// TwinCAT 3 PLC project RectangleSlicingMachine
// ProgramVersion: 3.1.4024.0
// libraries:
//   Tc2_MC2, * (Beckhoff Automation GmbH)
//   Tc2_NC, * (Beckhoff Automation GmbH)
//   Tc2_Standard, * (Beckhoff Automation GmbH)
//   Tc2_System, * (Beckhoff Automation GmbH)
//   Tc3_Module, * (Beckhoff Automation GmbH)
//   VisuDialogs, * (System)
// project tree:
//   / GlobalTextList.TcGTLO, PlcTask.TcTTO (not stored), Visualization Manager.TcVMO (not stored)
//   POUs/ FB_Slicer.TcPOU, MAIN.TcPOU, PRG_Test.TcPOU
//   VISUs/ Visualization.TcVIS
// real-time tasks:
//   TASK PlcTask: cycle T#10ms, priority 20, ADS port 350
// motion (NC):
//   TASK NC-Task 1 SAF: cycle T#2ms, priority 4, ADS port 501
//   TASK NC-Task 1 SVB: cycle T#10ms, priority 8, ADS port 511
//   AXIS AxisM1 (id 1)
//     General: UnitName=Degree
//     Velo: Maximum=18000
//     OtherSettings: AllowMotionCmdToSlave=true
//     encoder EncType=1
//     drive DrvType=5
//       Analog: TorqueSetpointScale=10, ScaleFactorActTorque=0.1
//       TimeComp: TaskDelayCycles=1
//     controller CtrType=1
//       CtrPara: PriorControlFactor=1
//         Observer: BandWidth=20
//   AXIS AxisM1s (id 2)
//     General: UnitName=Degree
//     Velo: Maximum=18000
//     OtherSettings: AllowMotionCmdToSlave=true
//     encoder EncType=1
//     drive DrvType=5
//       Analog: TorqueSetpointScale=10, ScaleFactorActTorque=0.1
//       TimeComp: TaskDelayCycles=1
//     controller CtrType=1
//       CtrPara: PriorControlFactor=1
//         Observer: BandWidth=20
//   AXIS AxisM2 (id 3)
//     General: UnitName=Degree
//     Velo: Maximum=18000
//     OtherSettings: AllowMotionCmdToSlave=true
//     encoder EncType=1
//     drive DrvType=5
//       Analog: TorqueSetpointScale=10, ScaleFactorActTorque=0.1
//       TimeComp: TaskDelayCycles=1
//     controller CtrType=1
//       CtrPara: PriorControlFactor=1
//         Observer: BandWidth=20
//   AXIS Axis 4 (id 4)
//     General: UnitName=°
//     Dynamic: Acceleration=12000, Deceleration=12000, Jerk=114759
//     Velo: Maximum=18000
//     PositionAreaControl: Enable=false
//     TargetPosControl: Enable=false
//     OtherSettings: AllowMotionCmdToSlave=true
//     encoder EncType=19
//       EncPara: ScaleFactorNumerator=360, ScaleFactorDenominator=65536, MaxCount=#xffffffff
//     drive DrvType=16
//       DrvPara: MaxCount=#xffffffff, DriveControlDWord=#x00020100
//         Analog: VeloReferenz=18000, TorqueSetpointScale=10, ScaleFactorActTorque=0.1
//         TimeComp: TaskDelayCycles=1
//     controller CtrType=1
//       CtrPara: PriorControlFactor=1
//         PosDiffControl: Enable=false
//         Observer: BandWidth=20
// I/O:
//   DEVICE Device 1 (EtherCAT) (disabled), AmsNetId 10.0.20.72.2.1
//     Drive 1 (i950 (BS-STO)) [i950 (BS-STO) FW V01.09]
//       modules: Module 1 (Universal (CSP + Speed and Torque Limits))
//     Drive 2 (i950 (BS-STO)) [i950 (BS-STO) FW V01.09]
//       modules: Module 1 (Universal (CSP + Speed and Torque Limits))
// variable links:
//   RectangleSlicingMachine/RectangleSlicingMachine Instance <-> Device 1 (EtherCAT)/Drive 1 (i950 (BS-STO))
//     PlcTask Outputs/MAIN.fbSlicer.nDrive1NegativeTorqueLimit <-> Module 1 (Universal (CSP + Speed and Torque Limits))/Torque Limits/MAIN.fbSlicer.nDrive1NegativeTorqueLimit
//     PlcTask Outputs/MAIN.fbSlicer.nDrive1PositiveTorqueLimit <-> Module 1 (Universal (CSP + Speed and Torque Limits))/Torque Limits/MAIN.fbSlicer.nDrive1PositiveTorqueLimit
//   RectangleSlicingMachine/RectangleSlicingMachine Instance <-> Device 1 (EtherCAT)/Drive 2 (i950 (BS-STO))
//     PlcTask Outputs/MAIN.fbSlicer.nDrive2NegativeTorqueLimit <-> Module 1 (Universal (CSP + Speed and Torque Limits))/Torque Limits/MAIN.fbSlicer.nDrive2NegativeTorqueLimit
//     PlcTask Outputs/MAIN.fbSlicer.nDrive2PositiveTorqueLimit <-> Module 1 (Universal (CSP + Speed and Torque Limits))/Torque Limits/MAIN.fbSlicer.nDrive2PositiveTorqueLimit
//   RectangleSlicingMachine/RectangleSlicingMachine Instance <-> NC-Task 1 SAF/Axes/AxisM1
//     PlcTask Inputs/MAIN.fbSlicer.AxisM1.NcToPlc <-> Outputs/ToPlc
//     PlcTask Outputs/MAIN.fbSlicer.AxisM1.PlcToNc <-> Inputs/FromPlc
//   RectangleSlicingMachine/RectangleSlicingMachine Instance <-> NC-Task 1 SAF/Axes/AxisM1s
//     PlcTask Inputs/MAIN.fbSlicer.AxisM1s.NcToPlc <-> Outputs/ToPlc
//     PlcTask Outputs/MAIN.fbSlicer.AxisM1s.PlcToNc <-> Inputs/FromPlc
//   RectangleSlicingMachine/RectangleSlicingMachine Instance <-> NC-Task 1 SAF/Axes/AxisM2
//     PlcTask Inputs/MAIN.fbSlicer.AxisM2.NcToPlc <-> Outputs/ToPlc
//     PlcTask Outputs/MAIN.fbSlicer.AxisM2.PlcToNc <-> Inputs/FromPlc

// ---- POUs/FB_Slicer.TcPOU
FUNCTION_BLOCK FB_Slicer
VAR_INPUT
	// Buttons to control various actions
	bStartButton : BOOL;
	bStopButton : BOOL;
	bContinueButton : BOOL;
	bHomeButton: BOOL;	// Returns axes to 0
	bEnginesOnButton : BOOL;
	bEnginesOffButton : BOOL;
	
	// Coordinates for the slicing start position
	aStartingPosition : ARRAY[0..1] OF LREAL;
	// Dimensions of the rectangle to be sliced
	aSlicingDimensions : ARRAY[0..1] OF LREAL;
	
	// Velocity override for motor movements
	fVelocityOverride : LREAL;
END_VAR
VAR_OUTPUT
	// Current positions of motors M1, M1s and M2
	fM1Position : LREAL;
	fM1sPosition : LREAL;
	fM2Position : LREAL;
	
	//Lights
	bEnginesLight : BOOL;	// On when the engines are on
	bHomedLight : BOOL;		// On when the axes are homed
	bSlicingLight : BOOL;	// On when slicing is happening
	bStopLight : BOOL;		// On when the process is stopped
	bErrorLight : BOOL;		// On when there's an error
	
	nErrorID : UDINT;
END_VAR
VAR
	// Trigger functions to stop bouncing when any of the buttons are pressed
	fbStartButtonTrigger : R_TRIG;
	fbStopButtonTrigger : R_TRIG;
	fbContinueButtonTrigger : R_TRIG;
	fbHomeButtonTrigger : R_TRIG;
	fbEnginesOnButtonTrigger : R_TRIG;
	fbEnginesOffButtonTrigger : R_TRIG;
	
	// References to the axes
	AxisM1 : AXIS_REF;	// Master
	AxisM1s : AXIS_REF;	// Slave
	AxisM2 : AXIS_REF;
	
	// Adequate function blocks needed for the axes
	M1McPower : MC_Power;
	M1McMoveRelative : MC_MoveRelative;
	M1McHome : MC_Home;
	M1McReset : MC_Reset;
	M1McStop : MC_Stop;
	
	M1sMcPower : MC_Power;
	M1sMcMoveRelative : MC_MoveRelative;
	M1sMcHome : MC_Home;
	M1sMcSetPosition : MC_SetPosition;
	M1sMcReset : MC_Reset;
	M1sMcStop : MC_Stop;
	
	M2McPower : MC_Power;
	M2McMoveRelative : MC_MoveRelative;
	M2McHome : MC_Home;
	M2McReset : MC_Reset;
	M2McStop : MC_Stop;
	
	// FBs needed to synchronise and desynchronize M1s to M1
	McGearIn : MC_GearIn;
	McGearOut : MC_GearOut;
	
	// Variable to tell us if the axes are homed or not
	bHomed : BOOL;
	
	// Variable to tell us if the engines are on or off (TRUE - ON, FALSE - OFF)
	bPowerStatus : BOOL;
	
	// Variable to tell us if M1 and M1s are coupled or not
	bCoupled  : BOOL;
	
	// Variable to tell us if the return button is pressed
	bReturned : BOOL;
	
	(* Variable to tell us if the user has given all coordinates needed (starting position and
	   rectangle dimensions) in order for the machine to be able to start *)
	bCoordinates : BOOL;
	
	// Variable to tell us if the dimensions we've given make the machine go out of bounds
	bLimit : BOOL;
	
	// Slicing dimensions 
	fM1SlicingDistance : LREAL;
	fM2SlicingDistance : LREAL;
	// Starting point dimensions
	fM1StartingDistance : LREAL;
	fM2StartingDistance : LREAL;
	
	// Variables used to keep track of the state in which we stopped and update the dimensions
	nStoppedState : DINT;
	fTempM1SlicingDistance : LREAL;
	fTempM2SlicingDistance : LREAL;
	fTempM1StartingDistance : LREAL;
	fTempM2StartingDistance : LREAL;

	
	// Variable needed for initializing the CASE structure states
	nCurrentState : DINT;
	
	// Needed torques for the I/O
	nDrive1PositiveTorqueLimit AT %Q* : INT := 1000;
    nDrive1NegativeTorqueLimit AT %Q* : INT := 1000;
    nDrive2PositiveTorqueLimit AT %Q* : INT := 1000;
    nDrive2NegativeTorqueLimit AT %Q* : INT := 1000;
	
END_VAR

VAR CONSTANT
	// Define limits
	MINIMUM_STARTING_POSITION : UINT := 10;
	MAXIMUM_SLICING_DIMENSION : UINT := 80;
END_VAR

(* This FB deals with controlling a machine that's got 3 motors with incremental encoders. Two of them (M1 & M1s) 
   function synchronous moving a slicer on the y axis whereas the third one (M2) moves the slicer on the x axis. 
   M1 & M1s have a master - slave configuration. The idea is that the machine will be used to cut rectangles with 
   dimensions given by the user, so what we want to do is to home the axes, take the slicer to a predefined 
   position where we want the slicing to start and cut out a rectangle by moving M1 & M1s synchronously positive 
   the y axis, then M2 in a positive direction on the x axis, then M1 & M1s negative y and then M2 negative x. 
   The machine operates within a 100x100cm workspace, which necessitates setting boundaries to avoid exceeding the 
   machine's limits. To ensure a safe margin, I've established a 10 cm buffer on all sides. So, the minimum starting
   position for any operation is (10,10) cm. Based on this configuration, the largest rectangle the machine can 
   safely cut is 80x80cm without crossing the predefined boundaries.*)
   
   
CASE nCurrentState OF
	0:	// Power OFF
	bEnginesLight := FALSE;
	bPowerStatus := FALSE;

	M1McPower.Enable := FALSE;
	M1McPower.Enable_Positive := FALSE;
	M1McPower.Enable_Negative := FALSE;
	M1McPower.Override := fVelocityOverride;
	
	M1sMcPower.Enable := FALSE;
	M1sMcPower.Enable_Positive := FALSE;
	M1sMcPower.Enable_Negative := FALSE;
	M1sMcPower.Override := fVelocityOverride;
	
	M2McPower.Enable := FALSE;
	M2McPower.Enable_Positive := FALSE;
	M2McPower.Enable_Negative := FALSE;
	M2McPower.Override := fVelocityOverride;
	  
	IF bEnginesOnButton THEN
		nCurrentState := 10;
	END_IF
	
	10:	// Power ON
	bEnginesLight := TRUE;
	bPowerStatus := TRUE;
	
	M1McPower.Enable := TRUE;
	M1McPower.Enable_Positive := TRUE;
	M1McPower.Enable_Negative := TRUE;
	M1McPower.Override := fVelocityOverride;
	
	M1sMcPower.Enable := TRUE;
	M1sMcPower.Enable_Positive := TRUE;
	M1sMcPower.Enable_Negative := TRUE;
	M1sMcPower.Override := fVelocityOverride;
	
	M2McPower.Enable := TRUE;
	M2McPower.Enable_Positive := TRUE;
	M2McPower.Enable_Negative := TRUE;
	M2McPower.Override := fVelocityOverride;
		  
	IF M1McPower.Active AND M1sMcPower.Active AND M2McPower.Active THEN
		nCurrentState := 25;
	END_IF		  

	25:	// Reseting
	bSlicingLight := FALSE;
	bStopLight := FALSE;
	
	// Reset the axes
	M1McReset.Execute := TRUE;
	IF NOT bCoupled THEN
		M1sMcReset.Execute := TRUE;
		IF M1sMcReset.Done THEN
			M1sMcReset.Execute := FALSE;
		END_IF
	END_IF
	M2McReset.Execute := TRUE;
	
	// If the reseting is done, go check if the axes are ready for operation
	IF M1McReset.Done AND M2McReset.Done THEN
		M1McReset.Execute := FALSE;	
		M2McReset.Execute := FALSE;
		
		//IF nStoppedState = 200 OR nStoppedState = 300 OR nStoppedState = 400 OR nStoppedState = 500 OR nStoppedState = 600 OR nStoppedState = 650 THEN
		//	nCurrentState := nStoppedState;
		//ELSE
		//	nCurrentState := 50;
		//END_IF
		
		nCurrentState := 50;
		
	END_IF
	
	// Check for errors during the reseting
	IF M1McReset.Error THEN
		nErrorID := M1McReset.ErrorID;
		nCurrentState := 999;
	END_IF
	IF M1sMcReset.Error THEN
		nErrorID := M1sMcReset.ErrorID;
		nCurrentState := 999;
	END_IF
	IF M2McReset.Error THEN
		nErrorID := M2McReset.ErrorID;
		nCurrentState := 999;
	END_IF

	50: // Checking if the axes are ready for operation
	IF M1McPower.Status AND M1sMcPower.Status AND M2McPower.Status AND bPowerStatus THEN
		nCurrentState := 75;
	END_IF	
	
	// If there is some error go to the error state
	IF M1McPower.Error THEN
		nErrorID := M1McPower.ErrorID;
		nCurrentState := 999;
	END_IF
	IF M1sMcPower.Error THEN
		nErrorID := M1sMcPower.ErrorID;
		nCurrentState := 999;
	END_IF
	IF M2McPower.Error THEN
		nErrorID := M2McPower.ErrorID;
		nCurrentState := 999;
	END_IF
	
	75:		// Setting the slave axis to 0
		M1sMcSetPosition.Execute := TRUE;
		M1sMcSetPosition.Position := 0;
					 
		IF M1sMcSetPosition.Done THEN
			M1sMcSetPosition.Execute := FALSE;
			nCurrentState := 100;
		END_IF

	100:	// Gearing
	// Synchronize M1s to M1. The ratio is 1 because they have to move synchronously
	McGearIn.Execute := TRUE;
	McGearIn.RatioNumerator := 1;
	McGearIn.RatioDenominator := 1;
		
	// If they're coupled go to homing
	IF McGearIn.InGear THEN
		bCoupled := TRUE;
		
		IF nStoppedState = 200 OR nStoppedState = 300 OR nStoppedState = 400 OR nStoppedState = 500 OR nStoppedState = 600 OR nStoppedState = 650 THEN
			nCurrentState := nStoppedState;
		ELSE
			nCurrentState := 150;
		END_IF
		
		//nCurrentState := 150;
	END_IF
	
	150:	// Homing
	// Home the axes with incremental encoders to 0
	M1McHome.Execute := TRUE;
	M1McHome.Position := 0;
	M1McHome.HomingMode := MC_Direct;
	
	M2McHome.Execute := TRUE;
	M2McHome.Position := 0;
	M2McHome.HomingMode := MC_Direct;
				 
	// If the homing is done, stop executing it
	IF M1McHome.Done AND M2McHome.Done THEN
		M1McHome.Execute := FALSE;
		M2McHome.Execute := FALSE;
	END_IF
	
	// If there is some error go to the error state
	IF M1McHome.Error THEN
		nErrorID := M1McHome.ErrorID;
		nCurrentState := 999;
	END_IF
	IF M2McHome.Error THEN
		nErrorID := M2McHome.ErrorID;
		nCurrentState := 999;
	END_IF
				
	// If the start button is pressed and the given coordinates are valid go to the slicing starting position 
	IF bStartButton AND bCoordinates THEN
		nCurrentState := 200;
	END_IF
	
	200:	// Slicing starting position
	IF nStoppedState = 200 THEN
		nStoppedState := 0;
		fM1StartingDistance := fTempM1StartingDistance;
		fM2StartingDistance := fTempM2StartingDistance;
	ELSE
		fTempM1StartingDistance := aStartingPosition[0];
		fTempM2StartingDistance := aStartingPosition[1];
	END_IF
	
	// Move all motors to the starting position
	M1McMoveRelative.Execute := TRUE;
	M1McMoveRelative.Distance := fTempM1StartingDistance;
	M1McMoveRelative.Velocity := 10;
	M1McMoveRelative.Acceleration := 10;
	M1McMoveRelative.Deceleration := 10;
	M1McMoveRelative.Jerk := 10000;
					 
	M2McMoveRelative.Execute := TRUE;
	M2McMoveRelative.Distance := fTempM2StartingDistance;
	M2McMoveRelative.Velocity := 10;
	M2McMoveRelative.Acceleration := 10;
	M2McMoveRelative.Deceleration := 10;
	M2McMoveRelative.Jerk := 10000;
					 
	// If all motors reach the starting position go to the first slicing state
	IF M1McMoveRelative.Done AND M2McMoveRelative.Done THEN
		M1McMoveRelative.Execute := FALSE;
		M2McMoveRelative.Execute := FALSE;
		
		nCurrentState := 300;
	END_IF
	
	// If error -> go to error state
	IF M1McMoveRelative.Error OR M2McMoveRelative.Error THEN
		IF M1McMoveRelative.Error THEN
			nErrorID := M1McMoveRelative.ErrorID;
		ELSIF M2McMoveRelative.Error THEN
			nErrorID := M2McMoveRelative.ErrorID;
		END_IF
		nCurrentState := 999;
	END_IF
					 
	300:	// Moving M1 & M1s positive y
	bSlicingLight := TRUE;
	
	IF nStoppedState = 300 THEN
		nStoppedState := 0;
		fM1SlicingDistance := fTempM1SlicingDistance;
	ELSE
		fM1SlicingDistance := aSlicingDimensions[0];
	END_IF
	
	M1McMoveRelative.Execute := TRUE;
	M1McMoveRelative.Distance := fM1SlicingDistance;
	M1McMoveRelative.Velocity := 5;
	M1McMoveRelative.Acceleration := 5;
	M1McMoveRelative.Deceleration := 5;
	M1McMoveRelative.Jerk := 10000;
				
	// If the moving is done, move on to the next	
	IF M1McMoveRelative.Done THEN
		M1McMoveRelative.Execute := FALSE;
		nCurrentState := 400;
	END_IF
	
	// If error -> go to error state
	IF M1McMoveRelative.Error THEN
		nErrorID := M1McMoveRelative.ErrorID;
		nCurrentState := 999;
	END_IF
	
	400:	// Moving M2 positive x
	bSlicingLight := TRUE;
	
	IF nStoppedState = 400 THEN
		nStoppedState := 0;
		fM2SlicingDistance := fTempM2SlicingDistance;
	ELSE
		fM2SlicingDistance := aSlicingDimensions[1];
	END_IF
	
	M2McMoveRelative.Execute := TRUE;
	M2McMoveRelative.Distance := fM2SlicingDistance;
	M2McMoveRelative.Velocity := 10;
	M2McMoveRelative.Acceleration := 10;
	M2McMoveRelative.Deceleration := 10;
	M2McMoveRelative.Jerk := 10000;
				
	// If the moving is done, move on to the next	
	IF M2McMoveRelative.Done THEN
		M2McMoveRelative.Execute := FALSE;
		nCurrentState := 500;
	END_IF
	
	// If error -> go to error state
	IF M2McMoveRelative.Error THEN
		nErrorID := M2McMoveRelative.ErrorID;
		nCurrentState := 999;
	END_IF
	
	500:	// Moving M1 & M1s negative y
	bSlicingLight := TRUE;
	
	IF nStoppedState = 500 THEN
		nStoppedState := 0;
		fM1SlicingDistance := fTempM1SlicingDistance;
	ELSE
		fM1SlicingDistance := aSlicingDimensions[0];
	END_IF
	
	M1McMoveRelative.Execute := TRUE;
	M1McMoveRelative.Distance := -fM1SlicingDistance;
	M1McMoveRelative.Velocity := 5;
	M1McMoveRelative.Acceleration := 5;
	M1McMoveRelative.Deceleration := 5;
	M1McMoveRelative.Jerk := 10000;
				
	// If the moving is done, move on to the next	
	IF M1McMoveRelative.Done THEN
		M1McMoveRelative.Execute := FALSE;
		nCurrentState := 600;
	END_IF
	
	// If error -> go to error state
	IF M1McMoveRelative.Error THEN
		nErrorID := M1McMoveRelative.ErrorID;
		nCurrentState := 999;
	END_IF
	
	600:	// Moving M2 negative x
	bSlicingLight := TRUE;
	
	IF nStoppedState = 600 THEN
		nStoppedState := 0;
		fM2SlicingDistance := fTempM2SlicingDistance;
	ELSE
		fM2SlicingDistance := aSlicingDimensions[1];
	END_IF
	
	M2McMoveRelative.Execute := TRUE;
	M2McMoveRelative.Distance := -fM2SlicingDistance;
	M2McMoveRelative.Velocity := 10;
	M2McMoveRelative.Acceleration := 10;
	M2McMoveRelative.Deceleration := 10;
	M2McMoveRelative.Jerk := 10000;
	
	// If the moving is done it means the rectangle is cut -> go to (0,0) position
	IF M2McMoveRelative.Done THEN
		M2McMoveRelative.Execute := FALSE;
		nCurrentState := 650;
	END_IF
	
	// If error -> go to error state
	IF M2McMoveRelative.Error THEN
		nErrorID := M2McMoveRelative.ErrorID;
		nCurrentState := 999;
	END_IF
	
	650:	// Return the axes to position (0,0)
	M1McMoveRelative.Execute := TRUE;
    M1McMoveRelative.Distance := -fM1Position;

    M2McMoveRelative.Execute := TRUE;
    M2McMoveRelative.Distance := -fM2Position;
	
	// If the axes are returned -> go to decouple the axes
	IF M1McMoveRelative.Done AND M2McMoveRelative.Done THEN
		M1McMoveRelative.Execute := FALSE;
		M2McMoveRelative.Execute := FALSE;
		nCurrentState := 700;
	END_IF
	
	// If error -> go to error state
	IF M1McMoveRelative.Error OR M2McMoveRelative.Error THEN
		IF M1McMoveRelative.Error THEN
			nErrorID := M1McMoveRelative.ErrorID;
		ELSIF M2McMoveRelative.Error THEN
			nErrorID := M2McMoveRelative.ErrorID;
		END_IF
		nCurrentState := 999;
	END_IF
	
	700:	// Decouple the axes
	McGearIn.Execute := FALSE;
			 
	McGearOut.Execute := TRUE;
			  
	// If the decoupling is done, move to the initial state
	IF McGearOut.Done THEN
		bCoupled := FALSE;
		McGearOut.Execute := FALSE;
				  
		IF NOT bEnginesLight THEN
			nCurrentState := 0;	  
		ELSE
			nCurrentState := 25;
		END_IF
	END_IF
	
	800:	// Stop	
	bSlicingLight := FALSE;
	bStopLight := TRUE;
	
	M1McStop.Execute := TRUE;
	M1McStop.Deceleration := 10;
	M1McStop.Jerk := 10000;
	
	M2McStop.Execute := TRUE;
	M2McStop.Deceleration := 10;
	M2McStop.Jerk := 10000;
			 
	IF M1McStop.Done THEN
		M1McStop.Execute := FALSE;
	END_IF
	
	IF M2McStop.Done THEN
		M2McStop.Execute := FALSE;
	END_IF
	
	// If we press on the continue button we want to continue where we left off
	IF bContinueButton THEN
		(* Since we are using incremental encoders and hence relative movements, we need 
		   to do some math to determine the distance the slicer should go to. We'll give these 
		   values as  dimensions of the rectangle or coordinates of the starting position. *)
		IF nStoppedState = 200 THEN
			fTempM1StartingDistance := aStartingPosition[0] - fM1Position;
			fTempM2StartingDistance := aStartingPosition[1] - fM2Position;
		ELSIF nStoppedState = 300 THEN
			fTempM1SlicingDistance := aStartingPosition[0] + aSlicingDimensions[0] - fM1Position;
		ELSIF nStoppedState = 400 THEN
			fTempM2SlicingDistance := aStartingPosition[1] + aSlicingDimensions[1] - fM2Position;
		ELSIF nStoppedState = 500 THEN
			fTempM1SlicingDistance := fM1Position - aStartingPosition[0];
		ELSIF nStoppedState = 600 THEN
			fTempM2SlicingDistance := fM2Position - aStartingPosition[1];
		END_IF
		
		nCurrentState := 700;	// Reseting must be done after stopping the axes
	END_IF
	
	IF bHomeButton THEN
		nStoppedState := 650;
		nCurrentState := 700;
	END_IF
	
	999:	// Error
	bErrorLight := TRUE;
	
	M1McStop.Execute := TRUE;
	M1McStop.Deceleration := 10;
	M1McStop.Jerk := 10000;
	
	M2McStop.Execute := TRUE;
	M2McStop.Deceleration := 10;
	M2McStop.Jerk := 10000;
			 
	IF M1McStop.Done THEN
		M1McStop.Execute := FALSE;
	END_IF
	
	IF M2McStop.Done THEN
		M2McStop.Execute := FALSE;
	END_IF
	
	ADSLOGDINT(msgCtrlMask := ADSLOG_MSGTYPE_ERROR,
			   msgFmtStr := TO_STRING(nErrorID),
			   dintArg := 0);
			   
	// If the start button is pressed go to the reset state 
	IF bStartButton THEN
		bErrorLight := FALSE;
		nCurrentState := 25;
	END_IF
END_CASE

// Trigger logic
fbStartButtonTrigger(CLK := bStartButton);
bStartButton := fbStartButtonTrigger.Q;
fbStopButtonTrigger(CLK := bStopButton);
bStopButton := fbStopButtonTrigger.Q;
fbContinueButtonTrigger(CLK := bContinueButton);
bContinueButton := fbContinueButtonTrigger.Q;
fbHomeButtonTrigger(CLK := bHomeButton);
bHomeButton := fbHomeButtonTrigger.Q;
fbEnginesOnButtonTrigger(CLK := bEnginesOnButton);
bEnginesOnButton := fbEnginesOnButtonTrigger.Q;
fbEnginesOffButtonTrigger(CLK := bEnginesOffButton);
bEnginesOffButton := fbEnginesOffButtonTrigger.Q;

// Stop the process if the stop button is pressed
IF bStopButton AND NOT bStopLight THEN
	M1McMoveRelative.Execute := FALSE;
	M2McMoveRelative.Execute := FALSE;
	nStoppedState := nCurrentState;
	nCurrentState := 800;
END_IF

(* If all current positions of the axes are 0 -> they're homed. I chose "<= 1" instead of "= 0"
   because I wanted to give some margin of error, ex. an axis being at a position of 0.02 *)
IF (fM1Position <= 1) AND (fM1sPosition <= 1) AND (fM2Position <= 1) THEN
	bHomedLight := TRUE;
	bHomed := TRUE;
ELSE
	bHomedLight := FALSE;
	bHomed := FALSE;
END_IF

// Home the axes if the return button is pressed
IF bHomeButton AND NOT bStopLight THEN
	// Reseting the stopped state if we want to home while stopped
	nStoppedState := 0;
	
	// We need to stop executing the movements first
	M1McMoveRelative.Execute := FALSE;
	M2McMoveRelative.Execute := FALSE;

	// I need to gear out first in order to be able to home the slave...
	nCurrentState := 700;
END_IF

IF bEnginesOffButton AND bHomed THEN
	bEnginesLight := FALSE;
	// Have to decouple the axis first because we can't home it if it's not decoupled
	nCurrentState := 700;
ELSIF bEnginesOffButton AND NOT bHomed THEN
	adslogdint(msgCtrlMask := ADSLOG_MSGTYPE_MSGBOX,
			   msgFmtStr := 'The process must be stopped and the axes must be homed before turning the engines off!',
			   dintArg := 0);
END_IF

(* This check ensures that the slicing operation stays within the 80x80 cm maximum allowed area 
   by comparing the sum of the starting position and slicing dimensions against the defined machine 
   boundaries. *)
IF aStartingPosition[0] + aSlicingDimensions[0] >  MINIMUM_STARTING_POSITION + MAXIMUM_SLICING_DIMENSION OR
   aStartingPosition[1] + aSlicingDimensions[1] > MINIMUM_STARTING_POSITION + MAXIMUM_SLICING_DIMENSION THEN
	bLimit := TRUE;
ELSE
	bLimit := FALSE;
END_IF

// Logic for the variable bCoordinates
IF aStartingPosition[0] = 0 OR aStartingPosition[1] = 0 OR 
   aStartingPosition[0] < MINIMUM_STARTING_POSITION OR 
   aStartingPosition[1] < MINIMUM_STARTING_POSITION OR
   aSlicingDimensions[0] = 0 OR aSlicingDimensions[1] = 0 OR
   aSlicingDimensions[0] > MAXIMUM_SLICING_DIMENSION OR 
   aSlicingDimensions[1] > MAXIMUM_SLICING_DIMENSION OR
   bLimit THEN
   
	bCoordinates := FALSE;
ELSE
	bCoordinates := TRUE;
END_IF

// Pop up boxes logic for when the start button is pressed but we can't start the process just yet
IF bStartButton THEN
	// If the engines are not turned on
	IF NOT bPowerStatus THEN
		adslogdint(msgCtrlMask := ADSLOG_MSGTYPE_MSGBOX,
			   msgFmtStr := 'The engines need to be turned on first!',
			   dintArg := 0);
	// If the axes are not homed
	ELSIF NOT bHomed THEN
		adslogdint(msgCtrlMask := ADSLOG_MSGTYPE_MSGBOX,
			   msgFmtStr := 'Axes need to be homed first!',
			   dintArg := 0);
	// If the limit is exceeded, indicate that the values are out of bounds
	ELSIF bLimit THEN
		adslogdint(msgCtrlMask := ADSLOG_MSGTYPE_MSGBOX,
			   msgFmtStr := 'Given values are out of bounds!',
			   dintArg := 0);
	// If coordinates for the starting position are not given
	ELSIF aStartingPosition[0] = 0 OR aStartingPosition[1] = 0 THEN
	adslogdint(msgCtrlMask := ADSLOG_MSGTYPE_MSGBOX,
			   msgFmtStr := 'You need to input coordinates for the starting position!',
			   dintArg := 0);
	// If the ooordinates are not valid
	ELSIF aStartingPosition[0] < MINIMUM_STARTING_POSITION OR aStartingPosition[1] < MINIMUM_STARTING_POSITION THEN
	adslogdint(msgCtrlMask := ADSLOG_MSGTYPE_MSGBOX,
			   msgFmtStr := 'Given coordinates are not valid! You need an input of at least 10!',
			   dintArg := 0);		
	// If slicing dimensions are not given
	ELSIF aSlicingDimensions[0] = 0 OR aSlicingDimensions[1] = 0 THEN
	adslogdint(msgCtrlMask := ADSLOG_MSGTYPE_MSGBOX,
			   msgFmtStr := 'You need to input the rectangle dimensions!',
			   dintArg := 0);
	// If the dimensions are not valid
	ELSIF aSlicingDimensions[0] > MAXIMUM_SLICING_DIMENSION OR aSlicingDimensions[1] > MAXIMUM_SLICING_DIMENSION THEN
	adslogdint(msgCtrlMask := ADSLOG_MSGTYPE_MSGBOX,
			   msgFmtStr := 'Given dimensions are not valid! You need inputs lower than or equal to (80, 80)!',
			   dintArg := 0);
	END_IF
END_IF

// Determine the current operating state of the axes 
AxisM1.ReadStatus();
AxisM1s.ReadStatus();
AxisM2.ReadStatus();

// Call instances of the MC FBs
M1McPower(Axis := AxisM1);
M1sMcPower(Axis := AxisM1s);
M2McPower(Axis := AxisM2);

M1McMoveRelative(Axis := AxisM1);
M1sMcMoveRelative(Axis := AxisM1s);
M2McMoveRelative(Axis := AxisM2);

M1McHome(Axis := AxisM1);
//M1sMcHome(Axis := AxisM1s);
M1sMcSetPosition(Axis := AxisM1s);
M2McHome(Axis := AxisM2);

M1McReset(Axis := AxisM1);
M1sMcReset(Axis := AxisM1s);
M2McReset(Axis := AxisM2);

M1McStop(Axis := AxisM1);
M1sMcStop(Axis := AxisM1s);
M2McStop(Axis := AxisM2);

McGearIn(Master := AxisM1, Slave := AxisM1s);
McGearOut(Slave := AxisM1s);

// Get the actual positions of each axis
fM1Position := AxisM1.NcToPlc.ActPos;
fM1sPosition := AxisM1s.NcToPlc.ActPos;
fM2Position := AxisM2.NcToPlc.ActPos;

END_FUNCTION_BLOCK

// ---- POUs/MAIN.TcPOU
PROGRAM MAIN
VAR
	fbSlicer : FB_Slicer;
	bStartButton : BOOL;
	bStopButton : BOOL;
	bContinueButton : BOOL;
	bHomeButton: BOOL;
	bEnginesOnButton : BOOL;
	bEnginesOffButton : BOOL;
	aStartingPosition : ARRAY[0..1] OF LREAL;
	aSlicingDimensions : ARRAY[0..1] OF LREAL;
	fVelocityOverride : LREAL := 80;
	fM1Position : LREAL;
	fM1sPosition : LREAL;
	fM2Position : LREAL;
	bEnginesLight : BOOL;
	bHomedLight : BOOL;
	bSlicingLight : BOOL;
	bStopLight : BOOL;
	bErrorLight : BOOL;
END_VAR

fbSlicer(bStartButton := bStartButton,
		 bStopButton := bStopButton,
		 bContinueButton := bContinueButton,
		 bHomeButton := bHomeButton,
		 bEnginesOnButton := bEnginesOnButton,
		 bEnginesOffButton := bEnginesOffButton,
		 aStartingPosition := aStartingPosition,
		 aSlicingDimensions := aSlicingDimensions,
		 fVelocityOverride := fVelocityOverride,
		 fM1Position => fM1Position,
		 fM1sPosition => fM1sPosition,
		 fM2Position => fM2Position,
		 bEnginesLight => bEnginesLight,
		 bHomedLight => bHomedLight,
		 bSlicingLight => bSlicingLight,
		 bStopLight => bStopLight,
		 bErrorLight => bErrorLight);
		 
//PRG_Test();

END_PROGRAM

// ---- POUs/PRG_Test.TcPOU
PROGRAM PRG_Test
VAR
	McPower : MC_Power;
	McHalt : MC_Halt;
	
	Axis : AXIS_REF;
	
	nCurrentState : DINT := 0;
	
	bPower : BOOL := FALSE;
	bHalt : BOOL := FALSE;
END_VAR

McPower(
	Axis:= Axis, 
	Enable:= bPower, 
	Enable_Positive:= TRUE, 
	Enable_Negative:= TRUE, 
	Override:= 100, 
	BufferMode:= , 
	Options:= , 
	Status=> , 
	Busy=> , 
	Error=> , 
	ErrorID=> );
	
McHalt(
	Axis:= Axis, 
	Execute:= bHalt, 
	Deceleration:= , 
	Jerk:= , 
	BufferMode:= , 
	Options:= , 
	Done=> , 
	Busy=> , 
	Active=> , 
	CommandAborted=> , 
	Error=> , 
	ErrorID=> );

END_PROGRAM

// ---- GlobalTextList.TcGTLO
TEXTLIST GlobalTextList
  162 = '%s'
  197 = 'Continue'
  569 = 'Engine Light'
  581 = 'Engines Off'
  318 = 'Engines On'
  598 = 'Error Light'
  570 = 'Home'
  667 = 'Homed Light'
  437 = 'length:'
  875 = 'Rectangle dimensions:'
  663 = 'Return'
  403 = 'Slicing dim'
  185 = 'Slicing Light'
  489 = 'Slicing pos'
  29 = 'Start'
  969 = 'Starting pos'
  599 = 'Starting position:'
  703 = 'Stop'
  651 = 'Stop Light'
  774 = 'Velocity override'
  468 = 'Velocity override:'
  302 = 'width:'
  196 = 'wifth:'
  3 = 'x:'
  674 = 'y:'
END_TEXTLIST

// ---- VISUs/Visualization.TcVIS
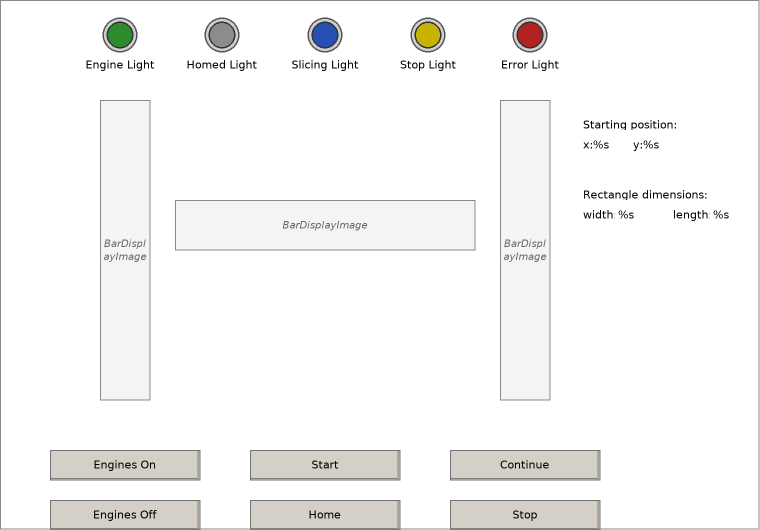
VISUALIZATION Visualization  // 760x530
    Button (250,450 150x30), "Start"
        tap MAIN.bStartButton
    BarDisplayImage (100,100 50x300), value: MAIN.fbSlicer.AxisM1.NcToPlc.ActPos, style: BarDisplayImage-Gray, scale format: %.1f, scale 0..100
    BarDisplayImage (500,100 50x300), value: MAIN.fbSlicer.AxisM1s.NcToPlc.ActPos, style: BarDisplayImage-Gray, scale format: %.1f, scale 0..100
    BarDisplayImage (175,200 300x50), value: MAIN.fbSlicer.AxisM2.NcToPlc.ActPos, style: BarDisplayImage-Gray, scale format: %.1f, scale 0..100
    Button (450,500 150x30), "Stop"
        tap MAIN.bStopButton
    Button (50,450 150x30), "Engines On"
        tap MAIN.bEnginesOnButton
    Button (50,500 150x30), "Engines Off"
        tap MAIN.bEnginesOffButton
    Button (250,500 150x30), "Home"
        tap MAIN.bHomeButton
    Lamp1 (100,15 40x40), variable: MAIN.bEnginesLight, style: Lamp-Lamp1-Green
    Lamp1 (202,15 40x40), variable: MAIN.bHomedLight, style: Lamp-Lamp1-Gray
    Lamp1 (305,15 40x40), variable: MAIN.bSlicingLight, style: Lamp-Lamp1-Blue
    Lamp1 (510,15 40x40), variable: MAIN.bErrorLight, style: Lamp-Lamp1-Red
    Label (80,50 80x30), "Engine Light"
    Label (182,50 80x30), "Homed Light"
    Label (285,50 80x30), "Slicing Light"
    Label (490,50 80x30), "Error Light"
    Rectangle (640,130 50x30), "%s", text variable: MAIN.aStartingPosition[0]
        OnMouseClick: write MAIN.aStartingPosition[0] via Default
    Label (580,110 150x30), "Starting position:"
    Rectangle (590,130 50x30), "%s", text variable: MAIN.aStartingPosition[1]
        OnMouseClick: write MAIN.aStartingPosition[1] via Default
    Label (580,180 150x30), "Rectangle dimensions:"
    Button (450,450 150x30), "Continue"
        tap MAIN.bContinueButton
    Lamp1 (408,15 40x40), variable: MAIN.bStopLight, style: Lamp-Lamp1-Yellow
    Label (388,50 80x30), "Stop Light"
    Label (630,130 20x30), "y:"
    Label (580,130 20x30), "x:"
    Label (670,200 50x30), "length:"
    Label (580,200 50x30), "width:"
    Rectangle (615,200 50x30), "%s", text variable: MAIN.aSlicingDimensions[1]
        OnMouseClick: write MAIN.aSlicingDimensions[1] via Default
    Rectangle (710,200 50x30), "%s", text variable: MAIN.aSlicingDimensions[0]
        OnMouseClick: write MAIN.aSlicingDimensions[0] via Default
END_VISUALIZATION
